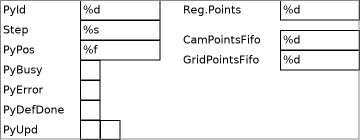
VISUALIZATION _VISU_ImageDeformation  // 360x140
VAR_IN_OUT
	m_Inst : FB_ImageDeformation;
END_VAR
    Rectangle (0,20 80x20), "Step"
    Rectangle (80,20 80x20), "%s", text variable: m_Inst._eDeformationStep
    Rectangle (0,40 80x20), "PyPos"
    Rectangle (80,40 80x20), "%f", text variable: m_Inst.fPythonPosition
    Rectangle (0,0 80x20), "PyId"
    Rectangle (80,0 80x20), "%d", text variable: m_Inst.nPythonId
    Rectangle (0,60 80x20), "PyBusy"
    RoundedRectangle (80,60 20x20), colour toggle: m_Inst.bPythonBusy
    Rectangle (0,80 80x20), "PyError"
    RoundedRectangle (80,80 20x20), colour toggle: m_Inst.bPythonError
    Rectangle (0,100 80x20), "PyDefDone"
    RoundedRectangle (80,100 20x20), colour toggle: m_Inst.bPythonDeformationDone
    Rectangle (0,120 80x20), "PyUpd"
    RoundedRectangle (80,120 20x20), tooltip "start update", colour toggle: m_Inst.bPythonStartUpdate
    RoundedRectangle (100,120 20x20), tooltip "update done", colour toggle: m_Inst.bPythonUpdateDone
    Rectangle (180,0 100x20), "Reg.Points"
    Rectangle (280,0 80x20), "%d", text variable: m_Inst._nCamPoints
    Rectangle (180,30 100x20), "CamPointsFifo"
    Rectangle (280,30 80x20), "%d", text variable: m_Inst.fbFifoCamPoints.nCount
    Rectangle (180,50 100x20), "GridPointsFifo"
    Rectangle (280,50 80x20), "%d", text variable: m_Inst.fbFifoGridPoints.nCount
END_VISUALIZATION

(* stored: Version 1.1.0.1, ProductVersion 3.1.4024.3
   Visu _VISU_ImageDeformation: Id {d7f8609f-6695-4ac1-9c58-fdd1ab1681e3} *)
